# EPICS autosave request: iocBoot/gmca_23i_ioc1/dbSave/assy.req
%
% BURT Request File
%
% $(ASSY)
%
$(ASSY):Start.DESC
$(ASSY):AccelTime
$(ASSY):AccelCurve
$(ASSY):Motion
